FUNCTION_BLOCK EL3214
VAR
	_io : EL3xx4_Data;
	{attribute addProperty Name "WcState"}
	_wcState : WcStateInputToggle;
	{attribute addProperty Name "Info data"}
	_infoData : InfoDataAds;
END_VAR

PROPERTY IO : REFERENCE TO EL3xx4_Data
GET
IO REF= _io;
END_GET
END_PROPERTY

PROPERTY WcState : REFERENCE TO WcStateInputToggle
GET
WcState REF= _wcState;
END_GET
END_PROPERTY

END_FUNCTION_BLOCK

(* stored: Version 1.1.0.1, ProductVersion 3.1.4024.9
   POU EL3214: Id {9e8e7aac-e9be-0465-2a1a-45fcb2dd12c7}, SpecialFunc None
   Property IO: Id {ac5dd1b5-5bc8-01e3-201d-8e1a819902e7}
   Get Get: Id {c2a9f534-afb5-054c-00f0-eea184064e51}
   Property WcState: Id {e21e3dec-e1c0-0a62-2dbf-8007cd109dc9}
   Get Get: Id {95361fb9-dd75-00e1-3cb7-fa99e5b10d36} *)
